(* CoDeSys 2.3 library: TcSUPS.lib *)
(* Libraries: STANDARD.LIB 5.6.98 13:03:02, TcBase.lib 14.5.09 13:14:08, TcSystem.lib*7.6.16 11:01:20, TcUtilities.lib*3.2.16 16:08:58 *)

(* Global variable list: Global_Seconds_UPS_Variables *)
VAR_GLOBAL
	eGlobalSUpsState	: E_S_UPS_State; (* current ups state of S-UPS *)
END_VAR
{library private}
VAR_GLOBAL CONSTANT
	BIOSIGRP_SUPS : UDINT := 16#00005000;
		BIOSIOFFS_SUPS_ENABLE					: UDINT := 16#00000000;	(* Enable/disable SUPS, W:1, R:0 *)
		BIOSIOFFS_SUPS_STATUS					: UDINT := 16#00000001;	(* SUPS status, W:0, R:1 *)
		BIOSIOFFS_SUPS_REVISION					: UDINT := 16#00000002;	(* SUPS revision, W:0, R:2 *)
		BIOSIOFFS_SUPS_SET_SHUTDOWN_TYPE		: UDINT := 16#00000005;	(* Set the Shutdown behavior, W:1, R:0 *)
		BIOSIOFFS_SUPS_GPIO_PIN 				: UDINT := 16#000000A0; (* Get the Address and the GPIO-Pin from PWR-Fail PIN, W:0, R:4 *)
		BIOSIOFFS_SUPS_GPIO_PIN_EX 				: UDINT := 16#000000A1; (* Get the Address and the GPIO-Pin from PWR-Fail PIN, W:0, R:24 *)
END_VAR
{library public}

(* Data type *)
TYPE E_S_UPS_Mode : (
	eSUPS_WrPersistData_Shutdown,			(* in case of powerfailure: writing of persistent data + shutdown*)
	eSUPS_WrPersistData_NoShutdown,			(* in case of powerfailure: writing of persistent data, no shutdown*)
	eSUPS_ImmediateShutdown,				(* in case of powerfailure: skips writing of data, immediate shutdown*)
	eSUPS_CheckPowerStatus					(* in case of powerfailure: reports powerfailure without action (no writing, no shutdown) *)
);
END_TYPE

(* Data type *)
TYPE E_S_UPS_State : (
	eSUPS_PowerOK,
	eSUPS_PowerFailure,
	eSUPS_WritePersistentData,
	eSUPS_QuickShutdown,
	eSUPS_WaitForRecover,
	eSUPS_WaitForPowerOFF
);


END_TYPE

(* POU F_GetVersionTcSUPS, ST *)
FUNCTION F_GetVersionTcSUPS : UINT	(* Gets the library version info *)
VAR_INPUT
	nVersionElement		:	INT;
(*
	Possible nVersionElement parameter:
	1	:	major number
	2	:	minor number
	3	:	revision number
*)
END_VAR
(* Version history:
Date			|	Version		|	created with				|	Author				|	Remark
dd.mm.yyyy	|					|								|						|
-----------------------------------------------------------------------------------------------------------------------------------------------------------------------------------------------------------------------------------------------------------------------------------
30.11.2009	|	1.0.0			|	TCAT2.11 B1539			|	I.Ch.				|	first release
15.01.2010	|	1.0.1			|	TCAT2.11 B1541			|	I.Ch.				|	global eGlobalSUpsState added
04.02.2011	|	1.0.2			|	TCAT2.11 B2024			|	I.Ch.				|	FB_S_UPS_EX added (extended functionality via BA-Lib)
04.02.2011	|	1.0.3			|	TCAT2.11 B2022			|	Christoph C		|	Debug code (functions/function blocks removed. BAVERSION_TO_DWORD function added.
04.02.2011	|	1.0.4			|	TCAT2.11 B2024			|	I.Ch.				|	BA version check updated
18.02.2011	|	1.0.5			|	TCAT2.11 B2024			|	Christoph C		|	Generic api function blocks, types and constants moved to the TcSystem.Lib, Small speed optimization of api function blocks.
21.05.2013	|	1.0.6			|	TCAT2.11 B2234			|	I.Ch.				|	BIOS-API-Version as internal but public variable in FB_S_UPS_EX; default powerfail reaction even if powerfail in first PLC cycle in FB_S_UPS
07.06.2016	|	1.0.7			|	TCAT2.11 B2256			|	I.Ch.				|	replaced FB_S_UPS_EX with FB_S_UPS_BAPI, unused internal POUs and DUTs removed
*)
CASE nVersionElement OF
1:	(* major number *)
	F_GetVersionTcSUPS := 1;
2:	(* minor number *)
	F_GetVersionTcSUPS := 0;
3:	(* revision number *)
	F_GetVersionTcSUPS := 7;
ELSE
	F_GetVersionTcSUPS := 16#FFFF;
END_CASE
END_FUNCTION

(* POU FB_NT_QuickShutdown, ST *)
FUNCTION_BLOCK FB_NT_QuickShutdown
VAR_INPUT
	NETID				:T_AmsNetId;
	START				:BOOL;
	TMOUT				:TIME := DEFAULT_ADS_TIMEOUT;
END_VAR
VAR_OUTPUT
	BUSY				:BOOL;
	ERR					:BOOL;
	ERRID				:UDINT;
END_VAR
{library private}
VAR
	ADSWRTCTL1			:ADSWRTCTL;
	RisingEdge			:R_TRIG;
	DELAY				:DWORD := 16#FFFFFFFF;
END_VAR
RisingEdge(CLK:=START);

IF RisingEdge.Q THEN
	ADSWRTCTL1(	NETID := NETID,
					PORT := AMSPORT_R3_SYSSERV,
					ADSSTATE := ADSSTATE_POWERFAILURE,
					DEVSTATE := 0,
					LEN := SIZEOF(DELAY),
					SRCADDR :=ADR(DELAY),
					Write := TRUE,
					TMOUT := TMOUT
				);
ELSE
	ADSWRTCTL1( Write:=FALSE);
END_IF


BUSY := ADSWRTCTL1.BUSY;
ERR := ADSWRTCTL1.ERR;
ERRID := ADSWRTCTL1.ERRID;
END_FUNCTION_BLOCK

(* POU FB_S_UPS, ST *)
FUNCTION_BLOCK FB_S_UPS
VAR_INPUT
	sNetID					: T_AmsNetId 		:= ''; 								(* '' = local netid *)
	iPLCPort				: UINT 				:= AMSPORT_R0_PLC_RTS1;				(* PLC Runtime System for writing persistent data *)
	iUPSPort				: UINT 				:= 16#4A8;							(* Port for reading Power State of UPS, dafault 16#4A8 *)
	tTimeout				: TIME 				:= DEFAULT_ADS_TIMEOUT;				(* ADS Timeout *)
	eUpsMode				: E_S_UPS_Mode		:= eSUPS_WrPersistData_Shutdown;	(* UPS mode (w/wo writing persistent data, w/wo shutdown) *)
	ePersistentMode			: E_PersistentMode	:= SPDM_2PASS;						(* mode for writing persistent data *)
	tRecoverTime			: TIME 				:= T#10s;							(* ON time to recover from short power failure in mode eSUPS_WrPersistData_NoShutdown/eSUPS_CheckPowerStatus  *)
END_VAR
VAR_OUTPUT
	bPowerFailDetect		: BOOL;													(* TRUE while powerfailure is detected *)
	eState					: E_S_UPS_State;										(* current ups state *)
END_VAR
{library private}
VAR
	fbWritePersistentData	: FB_WritePersistentData;
	fbNT_QuickShutdown 		: FB_NT_QuickShutdown;
	dwTemp					: DWORD;
	WaitForOffTimer			: TON;
	bFirstCycle				: BOOL := TRUE;
	bPowerOKInFirstCycle	: BOOL := FALSE;
END_VAR
(* monitor power state *)
dwTemp := FW_PortRead(iUPSPort, NoOfByte_DWord);
bPowerFailDetect := dwTemp.0;

(* load check *)
IF bFirstCycle THEN
	bFirstCycle 			:= FALSE;
	bPowerOKInFirstCycle 	:= NOT bPowerFailDetect;
END_IF

(* UPS State Machine *)
CASE eState OF
eSUPS_PowerOK:
	IF bPowerFailDetect THEN
		eState := eSUPS_PowerFailure; 		(* report powerfailure *)
		WaitForOffTimer(IN := FALSE, PT := tRecoverTime);
	END_IF


eSUPS_PowerFailure:
	IF bPowerOKInFirstCycle THEN
		(* allow saving/shutdown because S-UPS is fully loaded *)
		CASE eUpsMode OF
		eSUPS_WrPersistData_Shutdown,			(* in case of powerfailure: writing of persistent data + shutdown *)
		eSUPS_WrPersistData_NoShutdown:			(* in case of powerfailure: writing of persistent data, no shutdown *)
			(* start writing of persistent data *)
			fbWritePersistentData(
				NETID	:= sNetID,
				PORT	:= iPLCPort,
				START	:= TRUE,
				TMOUT	:= tTimeout,
				MODE	:= ePersistentMode
			);
			eState := eSUPS_WritePersistentData;


		eSUPS_CheckPowerStatus:					(* in case of powerfailure: reports powerfailure without action (no writing, no shutdown) *)
			(* check if power recovers *)
			eState := eSUPS_WaitForRecover;


		eSUPS_ImmediateShutdown:				(* in case of powerfailure: skips writing of data, immediate shutdown *)
			(* start quick shutdown *)
			fbNT_QuickShutdown(
				NETID := sNetID,
				START := TRUE,
				TMOUT := tTimeout
			);
			eState := eSUPS_QuickShutdown;

		END_CASE
	ELSE
		(* don't allow saving/shutdown because S-UPS was not fully loaded, just wait for recover or OFF *)
		eState := eSUPS_WaitForRecover;
	END_IF

eSUPS_WritePersistentData:
	(* writing of persistent data *)
	fbWritePersistentData(START	:= FALSE);

	IF eUpsMode = eSUPS_WrPersistData_NoShutdown THEN
		IF NOT fbWritePersistentData.BUSY THEN
			fbWritePersistentData(START	:= FALSE);

			(* wait for OFF *)
			eState := eSUPS_WaitForRecover;
			WaitForOffTimer(IN := FALSE, PT := tRecoverTime);
		END_IF
	ELSE
		IF NOT fbWritePersistentData.BUSY THEN
			fbWritePersistentData(START	:= FALSE);

			(* start quick shutdown *)
			fbNT_QuickShutdown(
				NETID := sNetID,
				START := TRUE,
				TMOUT := tTimeout
			);
			eState := eSUPS_QuickShutdown;
		END_IF
	END_IF


eSUPS_WaitForRecover:
	WaitForOffTimer(IN := (NOT bPowerFailDetect));
	IF WaitForOffTimer.Q THEN
		bPowerOKInFirstCycle := TRUE;
		eState := eSUPS_PowerOK; 		(* report powerOK *)
	END_IF


eSUPS_QuickShutdown:
	(* quick shutdown *)
	fbNT_QuickShutdown(START := FALSE);
	IF NOT fbNT_QuickShutdown.BUSY THEN
		fbNT_QuickShutdown(START := FALSE);

		(* wait for OFF *)
		eState := eSUPS_WaitForPowerOFF;
	END_IF


eSUPS_WaitForPowerOFF:
	(* wait for OFF *)
	eState := eSUPS_WaitForPowerOFF;

END_CASE

eGlobalSUpsState := eState;
END_FUNCTION_BLOCK

(* POU FB_S_UPS_BAPI, ST *)
FUNCTION_BLOCK FB_S_UPS_BAPI
VAR_INPUT
	sNetID					: T_AmsNetId 		:= ''; 								(* '' = local netid *)
	iPLCPort				: UINT;													(* PLC Runtime System for writing persistent data *)
	tTimeout				: TIME 				:= DEFAULT_ADS_TIMEOUT;				(* ADS Timeout *)
	eUpsMode				: E_S_UPS_Mode		:= eSUPS_WrPersistData_Shutdown;	(* UPS mode (w/wo writing persistent data, w/wo shutdown) *)
	ePersistentMode			: E_PersistentMode	:= SPDM_2PASS;						(* mode for writing persistent data *)
	tRecoverTime			: TIME 				:= T#10s;							(* ON time to recover from short power failure in mode eSUPS_WrPersistData_NoShutdown/eSUPS_CheckPowerStatus  *)
END_VAR
VAR_OUTPUT
	bPowerFailDetect		: BOOL;													(* TRUE while powerfailure is detected *)
	eState					: E_S_UPS_State := eSUPS_PowerOK;						(* current ups state *)
	nCapacity				: BYTE := 0;											(* actual capacity of UPS *)
	bBusy 					: BOOL;													(* TRUE: function block is busy *)
	bError 					: BOOL;													(* TRUE: function block has error *)
	nErrID 					: UDINT;												(* FB error ID   *)
END_VAR
{library private}
VAR
	fbSUpsGetGpioInfo		: FB_BaDeviceIoControl := ( nModifier := 0, affinity := ( lower := 0, higher := 0 ), nIdxGrp:=BIOSIGRP_SUPS, nIdxOffs:=BIOSIOFFS_SUPS_GPIO_PIN_EX );
	nSUpsGetGpioInfo		: DWORD;
	nGpioState				: INT;
	
	fbSUpsGetState			: FB_BaDeviceIoControl := ( nModifier := 0, affinity := ( lower := 0, higher := 0 ), nIdxGrp:=BIOSIGRP_SUPS, nIdxOffs:=BIOSIOFFS_SUPS_STATUS );
	nCapacityRsp			: BYTE;
	bCharging				: BOOL;
	bDischarging			: BOOL;
	nGetState				: INT;
	nUpsState				: INT;

	fbUpsStateTimer			: TON := (IN := TRUE);
	fbStartupTimer			: TON := (IN := TRUE, PT := T#0MS);
	nInitState				: INT;
	dxValue					: DWORD;
	dxStatus				: DWORD;
	dxBitMask				: DWORD;
	nBitNo 					: BYTE;
	bBitLevel				: BOOL;
	bStatus					: BOOL;
	bLowActive				: BOOL;
	bHighActive				: BOOL;
	bOldSupsVersion			: BOOL := TRUE;

	fbSUpsEnable			: FB_BaDeviceIoControl := ( nModifier := 0, affinity := ( lower := 0, higher := 0 ), nIdxGrp:=BIOSIGRP_SUPS, nIdxOffs:=BIOSIOFFS_SUPS_ENABLE );
	bSUps					: BOOL := TRUE;(* TRUE => enable S-UPS, FALSE => disable S-UPS *)
	bSUpsEnable				: BOOL := TRUE;
	nEnableState			: INT;

	fbSUpsGetRevision		: FB_BaDeviceIoControl := ( nModifier := 0, affinity := ( lower := 0, higher := 0 ), nIdxGrp:=BIOSIGRP_SUPS, nIdxOffs:=BIOSIOFFS_SUPS_REVISION );
	nSUpsVersionData		: ARRAY[0..2] OF BYTE;
	bSUpsGetRevision		: BOOL := TRUE;
	sSupsVersion			: STRING(15);
	nRevisionState			: INT;

	fbBaGenGetVersion		: FB_BaGenGetVersion;
	bBaGenGetVersion		: BOOL := TRUE;
	nVersion				: BYTE;
	nRevision				: BYTE;
 	nBuild					: WORD;
	sBaVersion				: STRING(15);
	bOldBaVersion			: BOOL := TRUE;

	bPowerFailDetectPrev	: BOOL;
	bPowerOKInFirstCycle	: BOOL;
	fbWritePersistentData	: FB_WritePersistentData;
	fbNT_QuickShutdown 		: FB_NT_QuickShutdown;
	WaitForOffTimer			: TON;
	bFirstCycle				: BOOL := TRUE;
END_VAR
VAR PERSISTENT
	bUseInfo				: BOOL;
	nIoAddr					: UDINT;
	nOffset					: BYTE;
	nParams					: BYTE;
	bUseInfoEx				: BOOL;
	stGpioInfoEx			: ST_WD_GPIO_InfoEx;
END_VAR
{library public}
(* initialization *)
CASE nInitState OF
0: 	
	IF NOT (bUseInfo OR bUseInfoEx) THEN
		fbStartupTimer(IN:= FALSE);
		nGpioState := 1;
		nInitState := 1;
	ELSIF bSUpsEnable THEN
		fbStartupTimer(IN:= FALSE);
		nEnableState := 1;
		nInitState := 2;
	ELSIF bSUpsGetRevision THEN
		fbStartupTimer(IN:= FALSE);
		nRevisionState := 1;
		nInitState := 3;
	ELSIF bBaGenGetVersion THEN
		fbStartupTimer(IN:= FALSE);
		nInitState := 4;
	END_IF

1:	(*get GPIO info*)
	fbStartupTimer(IN:= TRUE);
	IF fbStartupTimer.Q THEN
		fbStartupTimer(IN:= FALSE);

		CASE nGpioState OF
		1:
			bUseInfo	:= FALSE;
			nIoAddr		:= 0;
			nOffset 	:= 0;
			nParams 	:= 0;
			bUseInfoEx	:= FALSE;
			MEMSET(ADR(stGpioInfoEx), 0, SIZEOF(stGpioInfoEx));
			fbSUpsGetGpioInfo( bExecute := FALSE );
			fbSUpsGetGpioInfo( sNetID:=sNetID, cbWriteLen:= 0, cbReadLen:= SIZEOF(nSUpsGetGpioInfo), pWriteBuff:=0, pReadBuff:= ADR(nSUpsGetGpioInfo), bExecute:= TRUE, tTimeout:= tTimeout, nIdxOffs:=BIOSIOFFS_SUPS_GPIO_PIN );
			nGpioState := 2;
		2:	(*lagacy access*)
			fbSUpsGetGpioInfo( bExecute := FALSE );
			IF NOT fbSUpsGetGpioInfo.bBusy THEN
				IF NOT fbSUpsGetGpioInfo.bError THEN
					bUseInfo:= TRUE;
					nIoAddr	:= nSUpsGetGpioInfo AND 16#0000FFFF;
					nOffset := DWORD_TO_BYTE( DWORD#16#FF AND SHR( nSUpsGetGpioInfo, 16 ) );
					nParams := DWORD_TO_BYTE( DWORD#16#FF AND SHR( nSUpsGetGpioInfo, 24 ) );
					fbSUpsGetGpioInfo( bExecute := FALSE, bError=>bError, nErrID=>nErrID );
					fbStartupTimer(IN:= FALSE, PT := T#0MS);
					nGpioState := 0;
					nEnableState := 1;
					nInitState := nInitState + 1;
				ELSE
					IF ((UDINT_TO_DWORD(fbSUpsGetGpioInfo.nErrID) AND 16#0000FFFF) = 16#00000701) THEN
						fbSUpsGetGpioInfo( bExecute := FALSE );
						fbSUpsGetGpioInfo( sNetID:=sNetID, cbWriteLen:= 0, cbReadLen:= SIZEOF(stGpioInfoEx), pWriteBuff:=0, pReadBuff:= ADR(stGpioInfoEx), bExecute:= TRUE, tTimeout:= tTimeout, nIdxOffs:=BIOSIOFFS_SUPS_GPIO_PIN_EX );
						fbStartupTimer(IN:= FALSE, PT := T#100MS);
						nGpioState 	:= 3;
					ELSE
						fbSUpsGetGpioInfo( bExecute := FALSE, bError=>bError, nErrID=>nErrID );
						fbStartupTimer(IN:= FALSE, PT := T#100MS);
						nGpioState 	:= 0;
						nEnableState := 1;
						nInitState := nInitState + 1;
					END_IF
				END_IF
			END_IF
		3:	(*extended access*)
			fbSUpsGetGpioInfo( bExecute := FALSE);
			IF NOT fbSUpsGetGpioInfo.bBusy THEN
				IF NOT fbSUpsGetGpioInfo.bError THEN
					fbStartupTimer(IN:= FALSE, PT := T#0MS);
					bUseInfoEx := TRUE;
				ELSE
					fbStartupTimer(IN:= FALSE, PT := T#100MS);
				END_IF
				fbSUpsGetGpioInfo( bExecute := FALSE, bError=>bError, nErrID=>nErrID );
				nGpioState := 0;
				nEnableState := 1;
				nInitState := nInitState + 1;
			END_IF
		END_CASE
	END_IF
	
2:	(*enable UPS*)
	IF bSUpsEnable THEN
		fbStartupTimer(IN:= TRUE);
		IF fbStartupTimer.Q THEN
			fbStartupTimer(IN:= FALSE);

			CASE nEnableState OF
			1:
				fbSUpsEnable( bExecute := FALSE );
				fbSUpsEnable( sNetID:=sNetID, cbWriteLen:= SIZEOF(bSUps), cbReadLen:= 0, pWriteBuff:=ADR(bSUps), pReadBuff:= 0, bExecute:= TRUE, tTimeout:= tTimeout );
				nEnableState := 2;
			2:
				fbSUpsEnable( bExecute := FALSE, bError=>bError, nErrID=>nErrID );
				IF NOT fbSUpsEnable.bBusy THEN
					IF NOT fbSUpsEnable.bError THEN
						fbStartupTimer(IN:= FALSE, PT := T#0MS);
						bSUpsEnable := FALSE;
					ELSE
						fbStartupTimer(IN:= FALSE, PT := T#100MS);
					END_IF
					fbSUpsEnable( bExecute := FALSE );
					nEnableState := 0;
					nRevisionState := 1;
					nInitState := nInitState + 1;
				END_IF
			END_CASE
		END_IF
	ELSE
		nRevisionState := 1;
		nInitState := nInitState + 1;
	END_IF
	
3: 	(*get SPUS revision*)
	IF bSUpsGetRevision THEN
		fbStartupTimer(IN:= TRUE);
		IF fbStartupTimer.Q THEN
			fbStartupTimer(IN:= FALSE);
			
			CASE nRevisionState OF
			1:
				fbSUpsGetRevision( bExecute := FALSE );
				fbSUpsGetRevision( sNetID:=sNetID, cbWriteLen:= 0, cbReadLen:= SIZEOF(nSUpsVersionData), pWriteBuff:=0, pReadBuff:= ADR(nSUpsVersionData), bExecute:= TRUE, tTimeout:= tTimeout );
				nRevisionState := 2;
			2:
				fbSUpsGetRevision( bExecute := FALSE, bError=>bError, nErrID=>nErrID );
				IF NOT fbSUpsGetRevision.bBusy THEN
					IF NOT fbSUpsGetRevision.bError THEN
						sSupsVersion := CONCAT( BYTE_TO_STRING( nSUpsVersionData[0] ), CONCAT( '.', BYTE_TO_STRING( nSUpsVersionData[1] ) ) );
						bOldSupsVersion := (sSupsVersion > '0.0') AND (sSupsVersion < '1.5');
						fbStartupTimer(IN:= FALSE, PT := T#0MS);
						bSUpsGetRevision := FALSE;
					ELSE
						sSupsVersion := '';
						fbStartupTimer(IN:= FALSE, PT := T#100MS);
					END_IF
					fbSUpsGetRevision( bExecute := FALSE, bError=>bError, nErrID=>nErrID );
					nRevisionState := 0;
					nInitState := nInitState + 1;
				END_IF
			END_CASE
		END_IF
	ELSE
		nInitState := nInitState + 1;
	END_IF
	
4:	(*get BA version*)
	IF bBaGenGetVersion THEN
		fbStartupTimer(IN:= TRUE);
		IF fbStartupTimer.Q THEN
			fbStartupTimer(IN:= FALSE);
			fbBaGenGetVersion( sNetID:= '', bExecute:= TRUE );
	
			IF NOT fbBaGenGetVersion.bBusy THEN
				IF NOT fbBaGenGetVersion.bError THEN
					bBaGenGetVersion := FALSE;
					nVersion		:= fbBaGenGetVersion.nVersion;
					nRevision		:= fbBaGenGetVersion.nRevision;
					nBuild			:= fbBaGenGetVersion.nBuild;
					sBaVersion		:= CONCAT( CONCAT( CONCAT( CONCAT(BYTE_TO_STRING(nVersion), '.'), BYTE_TO_STRING(nRevision)), '.'), WORD_TO_STRING(nBuild));
					bOldBaVersion 	:= (BAVERSION_TO_DWORD(nVersion, nRevision, nBuild) < BAVERSION_TO_DWORD(1, 15, 0));
					fbStartupTimer(IN:= FALSE, PT := T#0MS);
				ELSE
					nVersion		:= 0;
					nRevision		:= 0;
					nBuild			:= 0;
					sBaVersion		:= '';
					bOldBaVersion 	:= FALSE;
					fbStartupTimer(IN:= FALSE, PT := T#100MS);
				END_IF
				fbBaGenGetVersion( bExecute:= FALSE, bError=>bError, nErrID=>nErrID );
				nInitState := 0;
			END_IF
		END_IF
	ELSE
		nInitState := 0;
	END_IF
END_CASE

(* monitor power state *)
IF bUseInfo THEN
	nBitNo 		:= SHR( nParams, 4 );(* higher nibble == bit number *)
	bBitLevel 	:= nParams.0;
	dxBitMask 	:= SHL( DWORD#16#1, nBitNo );(* create bit mask *)
	dxValue 	:= F_IOPortRead( nIoAddr + nOffset, NoOfByte_Byte );(* port read *)
	dxStatus 	:= dxValue AND dxBitMask;
	dxStatus 	:= SHR( dxStatus, nBitNo );
	bStatus		:= NOT ( dxStatus.0 XOR bBitLevel );
	bPowerFailDetect := bStatus; 

ELSIF bUseInfoEx THEN
	bLowActive 	:= NOT 	stGpioInfoEx.nFlags.3 AND NOT 	stGpioInfoEx.nFlags.2; (*00*)
	bHighActive := NOT 	stGpioInfoEx.nFlags.3 AND 		stGpioInfoEx.nFlags.2; (*01*)
	
	IF (stGpioInfoEx.nType = 0) AND (stGpioInfoEx.nLength = 4) AND ((bLowActive AND NOT bHighActive) OR (bHighActive AND NOT bLowActive)) THEN
		dxValue 	:= F_IOPortRead( stGpioInfoEx.nAddress, NoOfByte_DWord );(* port read *)
		dxBitMask 	:= stGpioInfoEx.nBitmask;
		bStatus 	:= ((dxValue AND dxBitMask) = dxBitMask);
		IF bHighActive THEN
			bPowerFailDetect := bStatus;
		ELSIF bLowActive THEN
			bPowerFailDetect := NOT bStatus;
		END_IF				
	ELSE
		(* not yet implemented *)
		nErrID	:= 16#701;
		bError	:= TRUE;
		bPowerFailDetect := FALSE;
	END_IF
END_IF

(* run *)
IF bFirstCycle THEN
	nCapacity := 0;
	IF iPLCPort = 0 THEN
		iPLCPort := (SystemInfo.runTimeNo-1) * 10 + 801; (*TwinCAT_SystemInfoVarList._AppInfo.AdsPort*);
	END_IF
	bFirstCycle := FALSE;
	bPowerOKInFirstCycle := NOT bPowerFailDetect;
END_IF

(* monitor charging state fast while < 90%, slow while >= 90% *)
fbUpsStateTimer();
IF fbUpsStateTimer.Q OR (bPowerFailDetect AND NOT bPowerFailDetectPrev) THEN
	IF bPowerFailDetect THEN
		fbUpsStateTimer.PT := T#50ms;
	ELSIF nCapacity >= 90 THEN
		fbUpsStateTimer.PT := T#1s;
	ELSE
		fbUpsStateTimer.PT := T#200ms;
	END_IF

	fbUpsStateTimer(IN := FALSE);
	fbUpsStateTimer(IN := TRUE);
	nGetState := 1;
END_IF

CASE nGetState OF
0:	(* idle *)
	;
1:
	fbSUpsGetState( bExecute := FALSE );
	fbSUpsGetState( sNetID:=sNetID, cbWriteLen:= 0, cbReadLen:= SIZEOF(nCapacityRsp), pWriteBuff:=0, pReadBuff:= ADR(nCapacityRsp), bExecute:= TRUE, tTimeout:= tTimeout );
	nGetState := 2;
2:
	fbSUpsGetState( bExecute := FALSE, bError=>bError, nErrID=>nErrID );
	IF NOT fbSUpsGetState.bBusy THEN
		IF NOT fbSUpsGetState.bError THEN
			IF ( ((nCapacityRsp >= 16#C0) AND (nCapacityRsp <= 16#CF)) OR ((nCapacityRsp >= 16#D0) AND (nCapacityRsp <= 16#DF)) ) THEN
				nUpsState := BYTE_TO_INT( nCapacityRsp AND 16#F0 );
				IF nUpsState = 16#C0 THEN
					bCharging := TRUE;
					bDischarging := FALSE;
				ELSIF nUpsState = 16#D0 THEN
					bCharging := FALSE;
					bDischarging := TRUE;
				ELSE
					bCharging := FALSE;
					bDischarging := FALSE;
				END_IF
				nCapacity := ( nCapacityRsp AND 16#0F ) * 10;
			ELSE
				nUpsState := nCapacityRsp;
				nCapacity := 0;
			END_IF
		ELSE
			nUpsState := 0;
			nCapacity := 0;
		END_IF
		fbSUpsGetState( bExecute := FALSE );
		nGetState := 0;
	END_IF
END_CASE

(* UPS State Machine *)
CASE eState OF
eSUPS_PowerOK:
	IF bPowerFailDetect THEN
		eState := eSUPS_PowerFailure; 		(* report powerfailure *)
		WaitForOffTimer(IN := FALSE, PT := tRecoverTime);
	END_IF

eSUPS_PowerFailure:
	IF bPowerOKInFirstCycle THEN
		(* allow saving/shutdown because S-UPS is fully loaded *)
		CASE eUpsMode OF
		eSUPS_WrPersistData_Shutdown,			(* in case of powerfailure: writing of persistent data + shutdown *)
		eSUPS_WrPersistData_NoShutdown:			(* in case of powerfailure: writing of persistent data, no shutdown *)
			IF (nCapacity >= 70) THEN
				(* start writing of persistent data *)
				fbWritePersistentData(
					NETID	:= sNetID,
					PORT	:= iPLCPort,
					START	:= TRUE,
					TMOUT	:= tTimeout,
					MODE	:= ePersistentMode
				);
				eState := eSUPS_WritePersistentData;
			ELSE
				(* don't allow saving/shutdown because S-UPS was not fully loaded *)
				IF eUpsMode = eSUPS_WrPersistData_NoShutdown THEN
					(* wait for OFF *)
					eState := eSUPS_WaitForRecover;
					WaitForOffTimer(IN := FALSE, PT := tRecoverTime);
				ELSE
					(* start quick shutdown *)
					fbNT_QuickShutdown(
						NETID := sNetID,
						START := TRUE,
						TMOUT := tTimeout
					);
					eState := eSUPS_QuickShutdown;
				END_IF
			END_IF

		eSUPS_CheckPowerStatus:					(* in case of powerfailure: reports powerfailure without action (no writing, no shutdown) *)
			(* check if power recovers *)
			eState := eSUPS_WaitForRecover;
	
		eSUPS_ImmediateShutdown:				(* in case of powerfailure: skips writing of data, immediate shutdown *)
			(* start quick shutdown *)
			nCapacity := 0;
			fbNT_QuickShutdown(
				NETID := sNetID,
				START := TRUE,
				TMOUT := tTimeout
			);
			eState := eSUPS_QuickShutdown;
		END_CASE

	ELSE
		(* don't allow saving/shutdown because S-UPS was not fully loaded, just wait for recover or OFF *)
		eState := eSUPS_WaitForRecover;
	END_IF

eSUPS_WritePersistentData:
	(* writing of persistent data *)
	fbWritePersistentData(START	:= FALSE);

	IF eUpsMode = eSUPS_WrPersistData_NoShutdown THEN
		IF NOT fbWritePersistentData.BUSY THEN
			fbWritePersistentData(START	:= FALSE);
			bError := fbWritePersistentData.ERR;
			nErrID := fbWritePersistentData.ERRID;

			(* wait for OFF *)
			eState := eSUPS_WaitForRecover;
			WaitForOffTimer(IN := FALSE, PT := tRecoverTime);
		END_IF
	ELSE
		IF NOT fbWritePersistentData.BUSY THEN
			fbWritePersistentData(START	:= FALSE);

			(* start quick shutdown *)
			fbNT_QuickShutdown(
				NETID := sNetID,
				START := TRUE,
				TMOUT := tTimeout
			);
			eState := eSUPS_QuickShutdown;
		END_IF
	END_IF

eSUPS_WaitForRecover:
	WaitForOffTimer(IN := (NOT bPowerFailDetect));
	IF NOT bPowerFailDetect THEN
		IF (nCapacity >= 90) OR WaitForOffTimer.Q THEN
			eState := eSUPS_PowerOK; 		(* report powerOK *)
			bPowerOKInFirstCycle := TRUE;
		END_IF
	END_IF

eSUPS_QuickShutdown:
	(* quick shutdown *)
	nCapacity := 0;
	fbNT_QuickShutdown(START := FALSE);
	IF NOT fbNT_QuickShutdown.BUSY THEN
		fbNT_QuickShutdown(START := FALSE);

		(* wait for OFF *)
		eState := eSUPS_WaitForPowerOFF;
	END_IF

eSUPS_WaitForPowerOFF:
	(* wait for OFF *)
	eState := eSUPS_WaitForPowerOFF;

END_CASE

bBusy := (nInitState <> 0) OR (nGetState <> 0) OR (eState = eSUPS_WritePersistentData) OR (eState = eSUPS_QuickShutdown);
eGlobalSUpsState := eState;
bPowerFailDetectPrev := bPowerFailDetect;
END_FUNCTION_BLOCK
